// TIA Portal V18 export
DATA_BLOCK "ST10_PMCountCycleTime"   // DB1061
{ S7_Optimized_Access := 'FALSE' }
// stored: AutoNumber false
   VAR
      PM : Array[1..30] of "RCS_CountCycleTime_V1";
      PM_Num : Int;
   END_VAR
BEGIN
END_DATA_BLOCK
